RoboDK station: TestStation.rdk

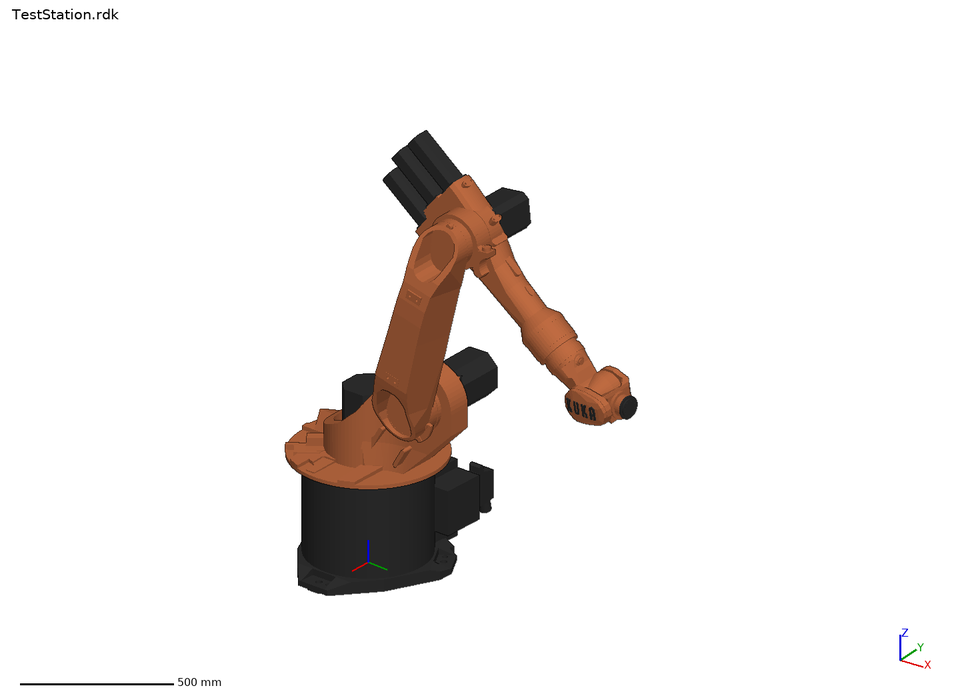
[picture v0: the station drawn from its stored meshes, robots at their saved joint values, targets as dots, program paths as lines]
Station TestStation (saved by RoboDK 5.6.0). Poses are relative to the parent item; angles as X-Y-Z fixed-axis rotations.
Station parameters (name, value as stored): LIN64
  - frame KUKA KR 16 2 Base at (0, 0, 0) mm, rotated rx 0 ry 0 rz -94.73 deg
    - robot KUKA KR 16 2: 6 axes, payload 16 kg, reach 1611 mm, repeatability 0.05 mm, weight 235 kg
        modified DH rows (alpha deg, a mm, theta deg, d mm): 0, 0, 0, 675; -90, 260, 0, 0; 0, 680, -90, 0; -90, -35, 0, 670; 90, 0, 0, 0; -90, 0, 180, 158
        joint limits [-185, -155, -130, -350, -130, -350] to [185, 35, 154, 350, 130, 350]; home [0, -90, 90, 0, 0, 0]; saved at [-91.98, -75.018, 113.959, -10.046, -42.435, 69.255]
      - tool Tool 1, TCP at (0, 0, 10) mm
  - Python program Kuka_Relative_Move_CoordCalc (listed below)

--- Python program Kuka_Relative_Move_CoordCalc ---
from robodk.robolink import *  # API to communicate with RoboDK
from robodk.robomath import *  # Robot toolbox
from robodk.robofileio import *

# Start communication with RoboDK
RDK = Robolink()

# Define the robot
ROBOT = RDK.ItemUserPick('Select a robot', ITEM_TYPE_ROBOT)
if not ROBOT.Valid():
    raise Exception('No robot selected or available')

# Specify the path to the CSV file
# csv_file = r'path_to_your_csv_file.csv'
# csv_file = r'C:\Users\paulo\OneDrive - Stellenbosch University\Masters\Thesis\3.Sim\Sim Verification\MovementFiles\test1.csv'
# csv_file = r'/home/paul/Downloads/test1.csv'
# csv_file = r'/home/paul/Sim_Analysis/Verification/MovMatrix.csv'
csv_file = r'/home/paul/FiducialTags/Simulations/Verification/Kuka_Files/MovMatrix_10.csv'

# csv_file = r'/test1.csv'

# Specify file codec
codec = 'utf-8'


initial_pose = ROBOT.Pose()
print(Mat(initial_pose))
target_ref = ROBOT.Pose()
pos_ref = target_ref.Pos()

# Load CSV data as a list of poses
def load_targets(strfile):
    csvdata = LoadList(strfile, ',', codec)
    poses = []
    for i in range(0, len(csvdata)):
        x, y, z, rx, ry, rz = csvdata[i][0:6]
        poses.append((x, y, z, rx, ry, rz))  # Store as a tuple

    return poses

# Move the robot to the poses from the CSV file
def move_robot_to_poses(strfile):
    poses = load_targets(strfile)

    # Set the robot's reference frame and tool frame
    ROBOT.setPoseFrame(ROBOT.PoseFrame())
    ROBOT.setPoseTool(ROBOT.PoseTool())
    # ROBOT.setG
    # Move the robot to the home position
    # ROBOT.MoveJ(ROBOT.JointsHome())

    # Move the robot to each pose from the CSV
    target_i = Mat(target_ref)
    for pose in poses:
        x, y, z, rx, ry, rz = pose  # Unpack the tuple
        # pose_matrix = transl(x, y, z) * rotz(rx * pi / 180) * roty(ry * pi / 180) * rotx(rx * pi / 180)
        # target_i = Offset(target_i, x,y,z,rx,ry,rz)
        target_i = RelTool(target_i, x, y, z, rx, ry, rz)

        # ROBOT.Pause(100000)
        ROBOT.MoveJ(target_i)


    ROBOT.MoveJ(initial_pose)

# Run the script to move the robot to the poses from the CSV file
move_robot_to_poses(csv_file)
